TYPE U_MOVE_DATA :
UNION
  stData              : ARRAY[1..MAX_MOVER] OF ST_MOVE_DATA;

  byData    AT %Q*    : ARRAY[1..MAX_MOVER] OF
                        ARRAY[1..SIZEOF(ST_MOVE_DATA)] OF BYTE;
END_UNION
END_TYPE

(* stored: Version 1.1.0.1
   DUT U_MOVE_DATA: Id {2c99304a-8c09-48cf-8bb1-9c319d233fee} *)
